PROGRAM PRG_PF1K2_WFS
VAR
    {attribute 'pytmc' := '
        pv: PF1K2:WFS
        io: io
    '}
    {attribute 'TcLinkTo' := '.fbThermoCouple1.bError 		:= TIIB[PF1K2-EL3314-E5]^TC Inputs Channel 1^Status^Error;
                              .fbThermoCouple1.bUnderrange	:= TIIB[PF1K2-EL3314-E5]^TC Inputs Channel 1^Status^Underrange;
                              .fbThermoCouple1.bOverrange 	:= TIIB[PF1K2-EL3314-E5]^TC Inputs Channel 1^Status^Overrange;
                              .fbThermoCouple1.iRaw 		:= TIIB[PF1K2-EL3314-E5]^TC Inputs Channel 1^Value;
                              .fbThermoCouple2.bError 		:= TIIB[PF1K2-EL3314-E5]^TC Inputs Channel 2^Status^Error;
                              .fbThermoCouple2.bUnderrange 	:= TIIB[PF1K2-EL3314-E5]^TC Inputs Channel 2^Status^Underrange;
                              .fbThermoCouple2.bOverrange 	:= TIIB[PF1K2-EL3314-E5]^TC Inputs Channel 2^Status^Overrange;
                              .fbThermoCouple2.iRaw 		:= TIIB[PF1K2-EL3314-E5]^TC Inputs Channel 2^Value'}
    fbPF1K2: FB_WFS;

    //stSiBP: ST_BeamParams := PMPS_GVL.cstFullBeam;
END_VAR

(*
   Avoid damage peak between 3.2 keV and 1.6 keV
*)
//stSiBp.neVRange := F_eVExcludeRange(1600, 3200);
// Drop transmission to 20%
//stSiBP.nTran := 0.2;

fbPF1K2.stOut.fPosition := -13.00;
fbPF1K2.stOut.bUseRawCounts := FALSE;
fbPF1K2.stOut.bValid := TRUE;
fbPF1K2.stOut.stPMPS.sPmpsState := 'PF1K2:WFS-OUT';

fbPF1K2.stTarget1.fPosition := -97.13;
fbPF1K2.stTarget1.bUseRawCounts := FALSE;
fbPF1K2.stTarget1.bValid := TRUE;
fbPF1K2.stTarget1.stPMPS.sPmpsState := 'PF1K2:WFS-TARGET1';

fbPF1K2.stTarget2.fPosition := -82.755;
fbPF1K2.stTarget2.bUseRawCounts := FALSE;
fbPF1K2.stTarget2.bValid := TRUE;
fbPF1K2.stTarget2.stPMPS.sPmpsState := 'PF1K2:WFS-TARGET2';

fbPF1K2.stTarget3.fPosition := -68.38;
fbPF1K2.stTarget3.bUseRawCounts := FALSE;
fbPF1K2.stTarget3.bValid := TRUE;
fbPF1K2.stTarget3.stPMPS.sPmpsState := 'PF1K2:WFS-TARGET3';

fbPF1K2.stTarget4.fPosition := -54.004;
fbPF1K2.stTarget4.bUseRawCounts := FALSE;
fbPF1K2.stTarget4.bValid := TRUE;
fbPF1K2.stTarget4.stPMPS.sPmpsState := 'PF1K2:WFS-TARGET4';

fbPF1K2.stTarget5.fPosition := -39.629;
fbPF1K2.stTarget5.bUseRawCounts := FALSE;
fbPF1K2.stTarget5.bValid := TRUE;
fbPF1K2.stTarget5.stPMPS.sPmpsState := 'PF1K2:WFS-TARGET5';

fbPF1K2(
    fbArbiter := GVL.fbArbiter2,
    fbFFHWO := GVL.fbFastFaultOutput2,
    stYStage := Main.M12,
    stZStage := Main.M13,
    sPmpsDeviceName := 'PF1K2:WFS',
    sTransitionKey := 'PF1K2:WFS-TRANSITION',
);

END_PROGRAM

(* stored: Version 1.1.0.1, ProductVersion 3.1.4022.18
   POU PRG_PF1K2_WFS: Id {46eac427-b476-476c-a121-178e6bb826c5}, SpecialFunc None *)
